// TIA Portal V16 export
// export: Created 2024-09-05T17:36:33.5824793Z, ExportSetting WithDefaults, DisplayName Totally Integrated Automation Portal, DisplayVersion V16 Update 6, DisplayName TIA Portal Version Control Interface, DisplayVersion V16 Update 2, DisplayName TIA Portal Openness, DisplayVersion V16 Update 6, DisplayName STEP 7 Professional, DisplayVersion V16 Update 6, DisplayName STEP 7 Safety, DisplayVersion V16, DisplayName WinCC Advanced, DisplayVersion V16 Update 6
VAR_GLOBAL   // PLC tag table "safety"
   iEmgStop AT %I1000.0 : Bool;
   iEmgStopDoors1 AT %I1000.1 : Bool;
   iEmgStopDoors2 AT %I1000.2 : Bool;
   iOpticalBarrier AT %I1010.0 : Bool;
   iTableInPosition AT %I1010.1 : Bool;
   iEmgStopOperatorII_HydraulicAgregate AT %I1010.2 : Bool;
   iStartCycle AT %I1010.3 : Bool;
   iEDM_KM20_KM21 AT %I1010.7 : Bool;
   iServiceMode AT %I1020.0 : Bool;
   iServiceDoorsLocked AT %I1020.2 : Bool;
   iSafetyScannerOK AT %I1020.1 : Bool;
   "q3L+" AT %Q2000.0 : Bool;   // emergency stop
   "q5L+" AT %Q2000.2 : Bool;   // emergency stop + service doors + light curtain
   "q4L+" AT %Q2000.1 : Bool;   // emergency stop + service doors
   iSafetyScannerReset AT %I1020.7 : Bool;
   "iEDM_A2.7_3L+" AT %I1100.0 : Bool;
   "iEDM_A2.8_4L+" AT %I1101.0 : Bool;
   "iEDM_A2.9_5L+" AT %I1102.0 : Bool;
   qRiveting1 AT %Q2010.0 : Bool;
   qRiveting2 AT %Q2010.1 : Bool;
   qServo1 AT %Q2010.2 : Bool;
   "q6L+" AT %Q2010.3 : Bool;   // valves on robot
   iServoSTOfeedback AT %I1000.7 : Bool;
   iEDM_KF101x AT %I1020.3 : Bool;
END_VAR
